% RSLogix 500 project PV9.RSS, saved by version 8.30.00.16 %
PROJECT "PV9"    % processor: Bul.1763 MicroLogix 1100 Series B %

PROGRAM FILES
  LAD 2   39 rungs

DATA FILES
  O0 OUTPUT  5 elements
  I1 INPUT  7 elements
  S2 STATUS  66 elements
  B3 BINARY  5 elements
  T4 TIMER  2 elements
  C5 COUNTER  1 elements
  R6 CONTROL  1 elements
  N7 INTEGER  1 elements
  F8 FLOAT  1 elements

LADDER 2
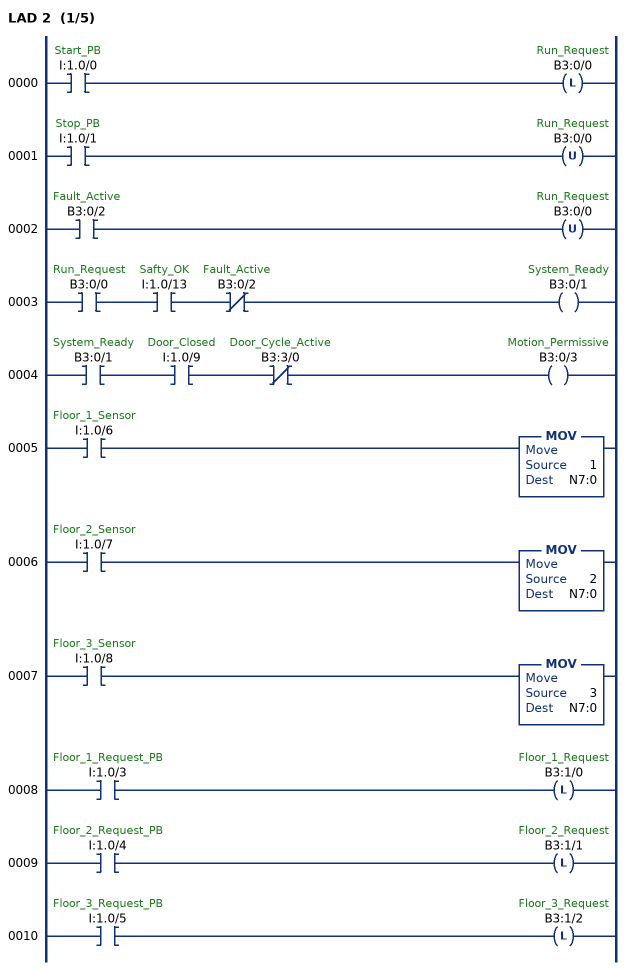
% Rung: 0 %
SOR XIC I:1.0/0 OTL B3:0/0 EOR
%   I:1.0/0  "Start_PB" %
%   B3:0/0  "Run_Request" %
% Rung: 1 %
SOR XIC I:1.0/1 OTU B3:0/0 EOR
%   I:1.0/1  "Stop_PB" %
%   B3:0/0  "Run_Request" %
% Rung: 2 %
SOR XIC B3:0/2 OTU B3:0/0 EOR
%   B3:0/2  "Fault_Active" %
%   B3:0/0  "Run_Request" %
% Rung: 3 %
SOR XIC B3:0/0 XIC I:1.0/13 XIO B3:0/2 OTE B3:0/1 EOR
%   B3:0/0  "Run_Request" %
%   I:1.0/13  "Safty_OK" %
%   B3:0/2  "Fault_Active" %
%   B3:0/1  "System_Ready" %
% Rung: 4 %
SOR XIC B3:0/1 XIC I:1.0/9 XIO B3:3/0 OTE B3:0/3 EOR
%   B3:0/1  "System_Ready" %
%   I:1.0/9  "Door_Closed" %
%   B3:3/0  "Door_Cycle_Active" %
%   B3:0/3  "Motion_Permissive" %
% Rung: 5 %
SOR XIC I:1.0/6 MOV 1 N7:0 EOR
%   I:1.0/6  "Floor_1_Sensor" %
% Rung: 6 %
SOR XIC I:1.0/7 MOV 2 N7:0 EOR
%   I:1.0/7  "Floor_2_Sensor" %
% Rung: 7 %
SOR XIC I:1.0/8 MOV 3 N7:0 EOR
%   I:1.0/8  "Floor_3_Sensor" %
% Rung: 8 %
SOR XIC I:1.0/3 OTL B3:1/0 EOR
%   I:1.0/3  "Floor_1_Request_PB" %
%   B3:1/0  "Floor_1_Request" %
% Rung: 9 %
SOR XIC I:1.0/4 OTL B3:1/1 EOR
%   I:1.0/4  "Floor_2_Request_PB" %
%   B3:1/1  "Floor_2_Request" %
% Rung: 10 %
SOR XIC I:1.0/5 OTL B3:1/2 EOR
%   I:1.0/5  "Floor_3_Request_PB" %
%   B3:1/2  "Floor_3_Request" %

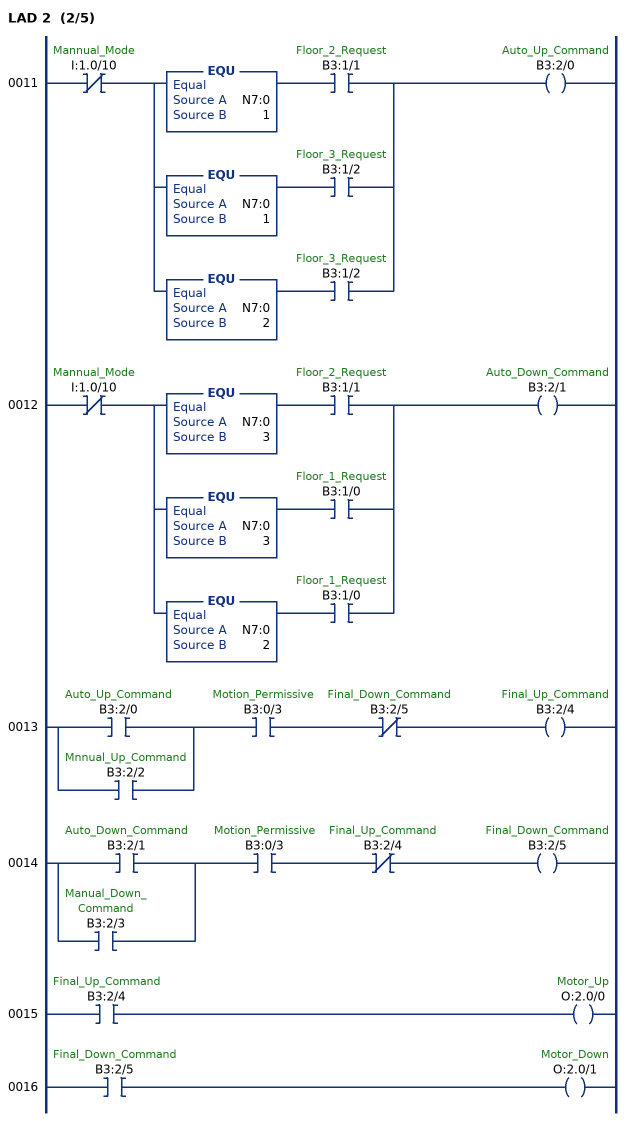
% Rung: 11 %
SOR XIO I:1.0/10 BST EQU N7:0 1 XIC B3:1/1 NXB BST EQU N7:0 1 XIC B3:1/2 NXB EQU N7:0 2 XIC B3:1/2 BND BND OTE B3:2/0 EOR
%   I:1.0/10  "Mannual_Mode" %
%   B3:1/1  "Floor_2_Request" %
%   B3:1/2  "Floor_3_Request" %
%   B3:2/0  "Auto_Up_Command" %
% Rung: 12 %
SOR XIO I:1.0/10 BST EQU N7:0 3 XIC B3:1/1 NXB BST EQU N7:0 3 XIC B3:1/0 NXB EQU N7:0 2 XIC B3:1/0 BND BND OTE B3:2/1 EOR
%   I:1.0/10  "Mannual_Mode" %
%   B3:1/1  "Floor_2_Request" %
%   B3:1/0  "Floor_1_Request" %
%   B3:2/1  "Auto_Down_Command" %
% Rung: 13 %
SOR BST XIC B3:2/0 NXB XIC B3:2/2 BND XIC B3:0/3 XIO B3:2/5 OTE B3:2/4 EOR
%   B3:2/0  "Auto_Up_Command" %
%   B3:2/2  "Mnnual_Up_Command" %
%   B3:0/3  "Motion_Permissive" %
%   B3:2/5  "Final_Down_Command" %
%   B3:2/4  "Final_Up_Command" %
% Rung: 14 %
SOR BST XIC B3:2/1 NXB XIC B3:2/3 BND XIC B3:0/3 XIO B3:2/4 OTE B3:2/5 EOR
%   B3:2/1  "Auto_Down_Command" %
%   B3:2/3  "Manual_Down_Command" %
%   B3:0/3  "Motion_Permissive" %
%   B3:2/4  "Final_Up_Command" %
%   B3:2/5  "Final_Down_Command" %
% Rung: 15 %
SOR XIC B3:2/4 OTE O:2.0/0 EOR
%   B3:2/4  "Final_Up_Command" %
%   O:2.0/0  "Motor_Up" %
% Rung: 16 %
SOR XIC B3:2/5 OTE O:2.0/1 EOR
%   B3:2/5  "Final_Down_Command" %
%   O:2.0/1  "Motor_Down" %

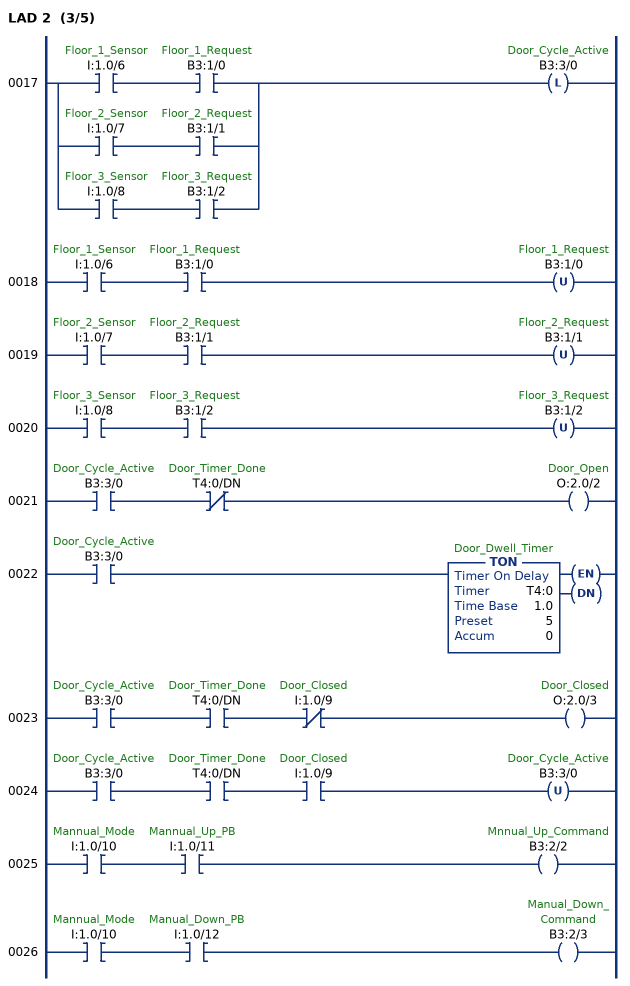
% Rung: 17 %
SOR BST XIC I:1.0/6 XIC B3:1/0 NXB BST XIC I:1.0/7 XIC B3:1/1 NXB XIC I:1.0/8 XIC B3:1/2 BND BND OTL B3:3/0 EOR
%   I:1.0/6  "Floor_1_Sensor" %
%   B3:1/0  "Floor_1_Request" %
%   I:1.0/7  "Floor_2_Sensor" %
%   B3:1/1  "Floor_2_Request" %
%   I:1.0/8  "Floor_3_Sensor" %
%   B3:1/2  "Floor_3_Request" %
%   B3:3/0  "Door_Cycle_Active" %
% Rung: 18 %
SOR XIC I:1.0/6 XIC B3:1/0 OTU B3:1/0 EOR
%   I:1.0/6  "Floor_1_Sensor" %
%   B3:1/0  "Floor_1_Request" %
% Rung: 19 %
SOR XIC I:1.0/7 XIC B3:1/1 OTU B3:1/1 EOR
%   I:1.0/7  "Floor_2_Sensor" %
%   B3:1/1  "Floor_2_Request" %
% Rung: 20 %
SOR XIC I:1.0/8 XIC B3:1/2 OTU B3:1/2 EOR
%   I:1.0/8  "Floor_3_Sensor" %
%   B3:1/2  "Floor_3_Request" %
% Rung: 21 %
SOR XIC B3:3/0 XIO T4:0/DN OTE O:2.0/2 EOR
%   B3:3/0  "Door_Cycle_Active" %
%   T4:0/DN  "Door_Timer_Done" %
%   O:2.0/2  "Door_Open" %
% Rung: 22 %
SOR XIC B3:3/0 TON T4:0 1.0 5 0 EOR
%   B3:3/0  "Door_Cycle_Active" %
%   T4:0  "Door_Dwell_Timer" %
% Rung: 23 %
SOR XIC B3:3/0 XIC T4:0/DN XIO I:1.0/9 OTE O:2.0/3 EOR
%   B3:3/0  "Door_Cycle_Active" %
%   T4:0/DN  "Door_Timer_Done" %
%   I:1.0/9  "Door_Closed" %
%   O:2.0/3  "Door_Closed" %
% Rung: 24 %
SOR XIC B3:3/0 XIC T4:0/DN XIC I:1.0/9 OTU B3:3/0 EOR
%   B3:3/0  "Door_Cycle_Active" %
%   T4:0/DN  "Door_Timer_Done" %
%   I:1.0/9  "Door_Closed" %
% Rung: 25 %
SOR XIC I:1.0/10 XIC I:1.0/11 OTE B3:2/2 EOR
%   I:1.0/10  "Mannual_Mode" %
%   I:1.0/11  "Mannual_Up_PB" %
%   B3:2/2  "Mnnual_Up_Command" %
% Rung: 26 %
SOR XIC I:1.0/10 XIC I:1.0/12 OTE B3:2/3 EOR
%   I:1.0/10  "Mannual_Mode" %
%   I:1.0/12  "Manual_Down_PB" %
%   B3:2/3  "Manual_Down_Command" %

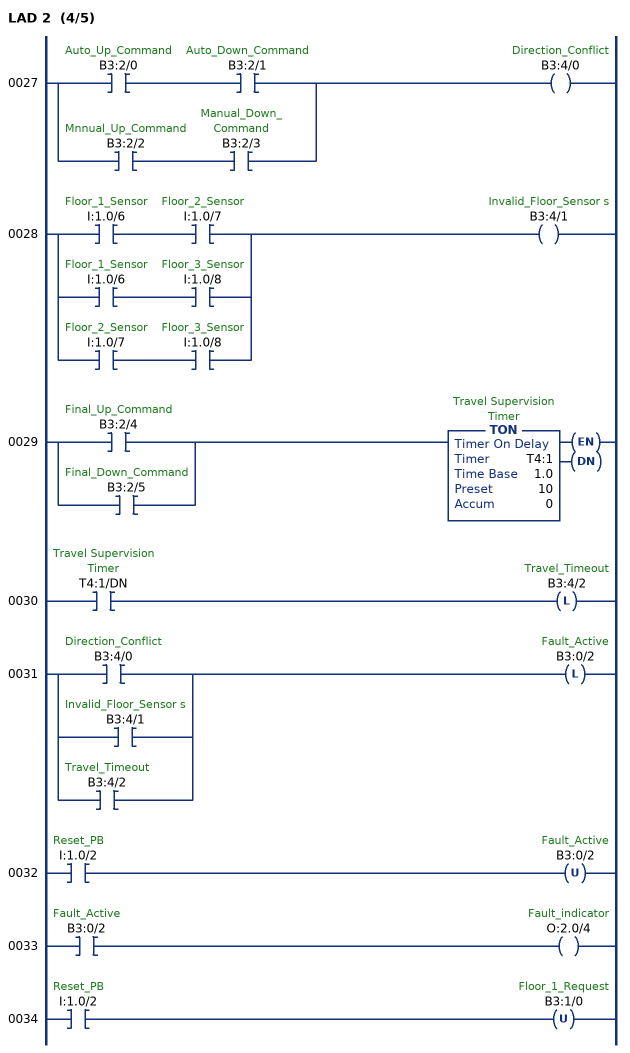
% Rung: 27 %
SOR BST XIC B3:2/0 XIC B3:2/1 NXB XIC B3:2/2 XIC B3:2/3 BND OTE B3:4/0 EOR
%   B3:2/0  "Auto_Up_Command" %
%   B3:2/1  "Auto_Down_Command" %
%   B3:2/2  "Mnnual_Up_Command" %
%   B3:2/3  "Manual_Down_Command" %
%   B3:4/0  "Direction_Conflict" %
% Rung: 28 %
SOR BST XIC I:1.0/6 XIC I:1.0/7 NXB BST XIC I:1.0/6 XIC I:1.0/8 NXB XIC I:1.0/7 XIC I:1.0/8 BND BND OTE B3:4/1 EOR
%   I:1.0/6  "Floor_1_Sensor" %
%   I:1.0/7  "Floor_2_Sensor" %
%   I:1.0/8  "Floor_3_Sensor" %
%   B3:4/1  "Invalid_Floor_Sensor s" %
% Rung: 29 %
SOR BST XIC B3:2/4 NXB XIC B3:2/5 BND TON T4:1 1.0 10 0 EOR
%   B3:2/4  "Final_Up_Command" %
%   B3:2/5  "Final_Down_Command" %
%   T4:1  "Travel Supervision Timer" %
% Rung: 30 %
SOR XIC T4:1/DN OTL B3:4/2 EOR
%   T4:1  "Travel Supervision Timer" %
%   B3:4/2  "Travel_Timeout" %
% Rung: 31 %
SOR BST XIC B3:4/0 NXB BST XIC B3:4/1 NXB XIC B3:4/2 BND BND OTL B3:0/2 EOR
%   B3:4/0  "Direction_Conflict" %
%   B3:4/1  "Invalid_Floor_Sensor s" %
%   B3:4/2  "Travel_Timeout" %
%   B3:0/2  "Fault_Active" %
% Rung: 32 %
SOR XIC I:1.0/2 OTU B3:0/2 EOR
%   I:1.0/2  "Reset_PB" %
%   B3:0/2  "Fault_Active" %
% Rung: 33 %
SOR XIC B3:0/2 OTE O:2.0/4 EOR
%   B3:0/2  "Fault_Active" %
%   O:2.0/4  "Fault_indicator" %
% Rung: 34 %
SOR XIC I:1.0/2 OTU B3:1/0 EOR
%   I:1.0/2  "Reset_PB" %
%   B3:1/0  "Floor_1_Request" %

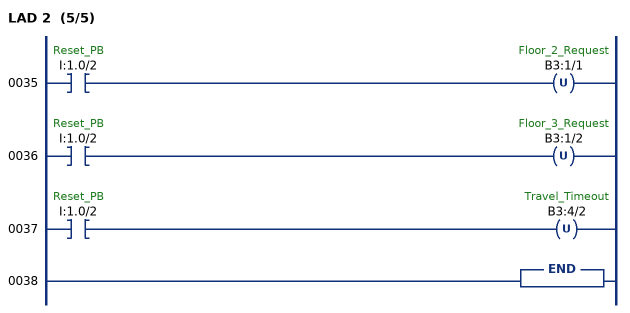
% Rung: 35 %
SOR XIC I:1.0/2 OTU B3:1/1 EOR
%   I:1.0/2  "Reset_PB" %
%   B3:1/1  "Floor_2_Request" %
% Rung: 36 %
SOR XIC I:1.0/2 OTU B3:1/2 EOR
%   I:1.0/2  "Reset_PB" %
%   B3:1/2  "Floor_3_Request" %
% Rung: 37 %
SOR XIC I:1.0/2 OTU B3:4/2 EOR
%   I:1.0/2  "Reset_PB" %
%   B3:4/2  "Travel_Timeout" %
% Rung: 38 %
SOR END EOR

DATA TABLE (non-zero values as saved)
DATA B3
% B3:0 % 0X000B 0X0000 0X0000 0X0000 0X0000
DATA T4
% .PRE .ACC %
% T4:0 % 5 0
% T4:1 % 10 0
DATA N7
% N7:0 % 1
